{attribute 'GeneratedUsingTerminal: ER5101-0002-0019'}
{attribute addProperty BoxType "ER5101-0002-0019"}
{attribute addProperty Id "ControlAT %Q*Control_D500AB792Set_counter_valueAT %Q*UINT2"}
{attribute addProperty CRC "3873217317"}
{attribute addProperty Size "4"}
TYPE ENC_Control_compact_E6DC9B25 EXTENDS OutputBase_10CEE7DE :
STRUCT
	{attribute addProperty Name "Control"}
	Control AT %Q* : Control_D500AB79;
	{attribute addProperty Name "Set_counter_value"}
	Set_counter_value AT %Q* : UINT;
END_STRUCT
END_TYPE

(* stored: Version 1.2.0.0, ProductVersion 3.1.4024.11
   DUT ENC_Control_compact_E6DC9B25: Id {91ccf89f-876d-4639-bd93-828d01749809} *)
